FUNCTION_BLOCK MUL_DINT (* IEC 61131-3 DINT Multiplication *)
  (* Standard: 61131-3 *)
  (* Version 0.0, 2004-12-15, JHC, Rockwell Automation, Converted from SRC format. *)
  (* Compiler header: package fb.rt.plc.math; *)
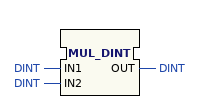
  VAR_INPUT
    IN1 : DINT; (* Multiplicand *)
    IN2 : DINT; (* Multiplier *)
  END_VAR
  VAR_OUTPUT
    OUT : DINT; (* Product *)
  END_VAR
END_FUNCTION_BLOCK
